// TIA Portal project "2022.06.05_比较操作2" (V17)

(* hardware
DEVICE "S7-1200 station_1"  S7-1200 Station
   slot 0: "Rack_0"  S7-1200 Rack  Rack  V1.0
   slot 1: "PLC_1"  CPU 1212C DC/DC/DC  6ES7 212-1AE40-0XB0  V4.5
*)

// ===== PLC "PLC_1"  CPU 1212C DC/DC/DC =====

VAR_GLOBAL   // PLC tag table "默认变量表"
   "Tag_1" AT %I0.0 : Bool;
   "标志位" AT %M0.0 : Bool;
   "故障" AT %I0.2 : Bool;
   "Tag_4" AT %MW10 : Int;
   "红" AT %Q0.0 : Bool;
   "启动" AT %I0.1 : Bool;
   "初始位" AT %M1.0 : Bool;
   "Tag_2" AT %M0.1 : Bool;
   "赋值" AT %I0.3 : Bool;
   "Tag_7" AT %I0.4 : Bool;
   "加" AT %I0.5 : Bool;
   "Tag_9" AT %M10.0 : Bool;
   "减" AT %I0.6 : Bool;
   "手动复位(1)" AT %I0.7 : Bool;
   "Tag_12" AT %M10.1 : Bool;
   "当前值" AT %MW20 : Int;
   "Tag_6" AT %M0.2 : Bool;
   "5次" AT %M0.3 : Bool;
   "绿和闪" AT %Q0.1 : Bool;
   "黄" AT %Q0.2 : Bool;
   "Tag_3" AT %MW0 : Int;
   "Tag_8" AT %Q0.3 : Bool;
   "Tag_10" AT %Q0.4 : Bool;
   "当前时间" AT %MD100 : DWord;
   "System_Byte" AT %MB1 : Byte;
   "FirstScan" AT %M1.0 : Bool;
   "DiagStatusUpdate" AT %M1.1 : Bool;
   "AlwaysTRUE" AT %M1.2 : Bool;
   "AlwaysFALSE" AT %M1.3 : Bool;
   "Clock_Byte" AT %MB20 : Byte;
   "Clock_10Hz" AT %M20.0 : Bool;
   "Clock_5Hz" AT %M20.1 : Bool;
   "Clock_2.5Hz" AT %M20.2 : Bool;
   "Clock_2Hz" AT %M20.3 : Bool;
   "Clock_1.25Hz" AT %M20.4 : Bool;
   "Clock_1Hz" AT %M20.5 : Bool;
   "Clock_0.625Hz" AT %M20.6 : Bool;
   "Clock_0.5Hz" AT %M20.7 : Bool;
   "急停" AT %I1.0 : Bool;
END_VAR

// folder: System blocks/Program resources

DATA_BLOCK "IEC_Counter_0_DB"   // DB1
{ S7_Optimized_Access := 'TRUE' }
AUTHOR : Simatic
FAMILY : IEC
NAME : CNTR
VERSION : 1.0
// stored: InstanceOfName IEC_COUNTER
"IEC_COUNTER"
BEGIN
END_DATA_BLOCK

DATA_BLOCK "IEC_Counter_0_DB_1"   // DB2
{ S7_Optimized_Access := 'TRUE' }
AUTHOR : Simatic
FAMILY : IEC
NAME : CNTR
VERSION : 1.0
// stored: InstanceOfName IEC_COUNTER
"IEC_COUNTER"
BEGIN
END_DATA_BLOCK

DATA_BLOCK "IEC_Counter_0_DB_2"   // DB3
{ S7_Optimized_Access := 'TRUE' }
AUTHOR : Simatic
FAMILY : IEC
NAME : CNTR
VERSION : 1.0
// stored: InstanceOfName IEC_COUNTER
"IEC_COUNTER"
BEGIN
END_DATA_BLOCK

DATA_BLOCK "IEC_Timer_0_DB"   // DB4
{ S7_Optimized_Access := 'TRUE' }
AUTHOR : Simatic
FAMILY : IEC
NAME : IEC_TMR
VERSION : 1.0
// stored: InstanceOfName IEC_TIMER
"IEC_TIMER"
BEGIN
END_DATA_BLOCK

DATA_BLOCK "IEC_Counter_0_DB_3"   // DB5
{ S7_Optimized_Access := 'TRUE' }
AUTHOR : Simatic
FAMILY : IEC
NAME : CNTR
VERSION : 1.0
// stored: InstanceOfName IEC_COUNTER
"IEC_COUNTER"
BEGIN
END_DATA_BLOCK

DATA_BLOCK "IEC_Counter_0_DB_4"   // DB6
{ S7_Optimized_Access := 'TRUE' }
AUTHOR : Simatic
FAMILY : IEC
NAME : CNTR
VERSION : 1.0
// stored: InstanceOfName IEC_COUNTER
"IEC_COUNTER"
BEGIN
END_DATA_BLOCK

DATA_BLOCK "IEC_Timer_0_DB_1"   // DB7
{ S7_Optimized_Access := 'TRUE' }
AUTHOR : Simatic
FAMILY : IEC
NAME : IEC_TMR
VERSION : 1.0
// stored: InstanceOfName IEC_TIMER
"IEC_TIMER"
BEGIN
END_DATA_BLOCK

// folder: (top level)

ORGANIZATION_BLOCK "Main"   // OB1, LAD, ProgramCycle
TITLE = "Main Program Sweep (Cycle)"
{ S7_Optimized_Access := 'TRUE' }
VERSION : 0.1
   VAR_INPUT
      Initial_Call : Bool;   // Initial call of this OB
      Remanence : Bool;   // =True, if remanent data are available
   END_VAR
   VAR_TEMP   // added for the SCL form of the ladder/FBD networks
      _w1 : Bool;
   END_VAR
BEGIN

REGION Network 1
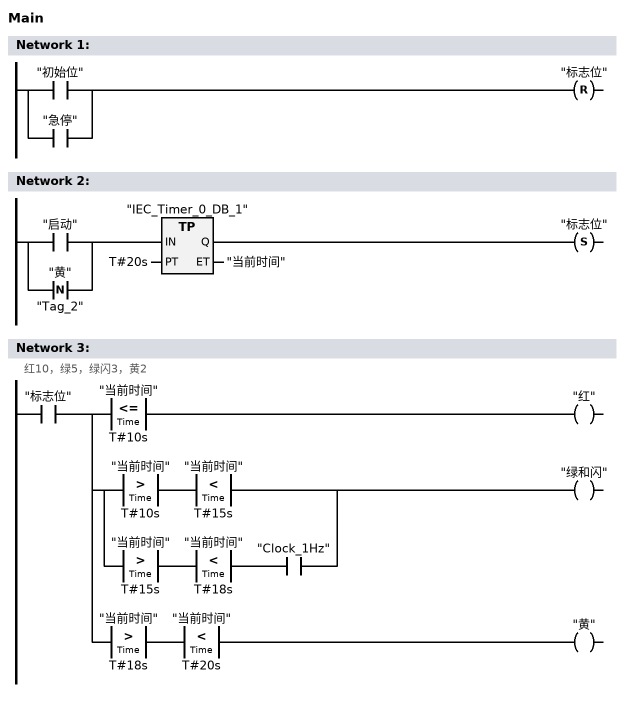
   RUNG wire#powerrail
      Contact( "初始位" )
      wire#w1
      R_Coil( "标志位" )
   END_RUNG
   RUNG wire#powerrail
      Contact( "急停" )
   END_RUNG wire#w1
   // the same network as SCL:
   IF "初始位" OR "急停" THEN "标志位" := FALSE; END_IF;
END_REGION

REGION Network 2
   #_w1 := NOT "黄" AND "Tag_2";   // falling edge of "黄"
   "Tag_2" := "黄";
   "IEC_Timer_0_DB_1".TP(IN := "启动" OR #_w1, PT := T#20s, ET => "当前时间");
   IF "IEC_Timer_0_DB_1".Q THEN "标志位" := TRUE; END_IF;
END_REGION

REGION Network 3
   // 红10，绿5，绿闪3，黄2
   RUNG wire#powerrail
      Contact( "标志位" )
      wire#w1
      { S7_Templates := "SrcType := Time" } LE_Contact(in1 := "当前时间", in2 := T#10s)
      Coil( "红" )
   END_RUNG
   RUNG wire#w1
      { S7_Templates := "SrcType := Time" } GT_Contact(in1 := "当前时间", in2 := T#10s)
      { S7_Templates := "SrcType := Time" } LT_Contact(in1 := "当前时间", in2 := T#15s)
      wire#w2
      Coil( "绿和闪" )
   END_RUNG
   RUNG wire#w1
      { S7_Templates := "SrcType := Time" } GT_Contact(in1 := "当前时间", in2 := T#15s)
      { S7_Templates := "SrcType := Time" } LT_Contact(in1 := "当前时间", in2 := T#18s)
      Contact( "Clock_1Hz" )
   END_RUNG wire#w2
   RUNG wire#w1
      { S7_Templates := "SrcType := Time" } GT_Contact(in1 := "当前时间", in2 := T#18s)
      { S7_Templates := "SrcType := Time" } LT_Contact(in1 := "当前时间", in2 := T#20s)
      Coil( "黄" )
   END_RUNG
   // the same network as SCL:
   "红" := "标志位" AND ("当前时间" <= T#10s);
   "绿和闪" := "标志位" AND ((("当前时间" > T#10s) AND ("当前时间" < T#15s)) OR (("当前时间" > T#15s) AND ("当前时间" < T#18s) AND "Clock_1Hz"));
   "黄" := "标志位" AND ("当前时间" > T#18s) AND ("当前时间" < T#20s);
END_REGION
END_ORGANIZATION_BLOCK